TYPE ST_OvercurrentProtection_get :
STRUCT
	//Overcurrent Powerlocks
	r_TotalOutputCurrentLimit			: REAL := 0;
	r_TotalInputCurrentLimit			: REAL := 0;
	b_OutputWarning						: BOOL;
	b_InputWarning						: BOOL;
	b_OutputAlarm						: BOOL;
	b_InputAlarm						: BOOL;
	r_PeakCurrent						: REAL;
	t_PeakCurrentDuration				: TIME;
	s_locationPeak						: STRING;
	
	Events								: ST_OvercurrentProtection_events;
END_STRUCT
END_TYPE

(* stored: Version 1.1.0.1, ProductVersion 3.1.4026.18
   DUT ST_OvercurrentProtection_get: Id {5d76d2f2-7ee8-483d-8121-a381449661f0} *)
